Staubli VAL3: remGetMaxDist.pgx

program remGetMaxDist(string& sReturn[] (dimensions=1))
  local string sCmd
begin
  // Return max dist in a single move step for remote moves (mm)
  //
  logMsg("call remGetMaxDist")
  sCmd="GETMAXDIST"
  call remGetnGlobal(nMaxAccel,sCmd,sReturn)
end
